// Mitsubishi GX Works2 project: sw1-4   PLC: FX1N/FX1NC

PROGRAM MAIN
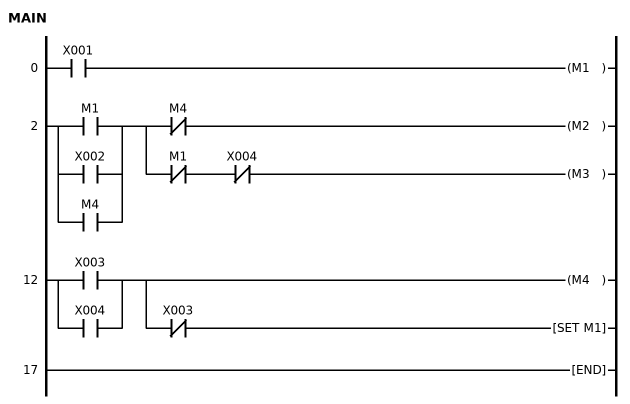
0     LD      X001
      OUT     M1
2     LD      M1
      OR      X002
      OR      M4
      MPS
      ANI     M4
      OUT     M2
      MPP
      ANI     M1
      ANI     X004
      OUT     M3
12    LD      X003
      OR      X004
      OUT     M4
      ANI     X003
      SET     M1
17    END
END_PROGRAM
